Fanuc KAREL source: wcartfltrenb.kl

PROGRAM wcartfltrenb
%NOLOCKGROUP
VAR
  p : POSITION
  q : POSITION
  i : INTEGER
  r : REAL
BEGIN
  WITH $CARTFLTRENB = TRUE MOVE TO p
END wcartfltrenb
